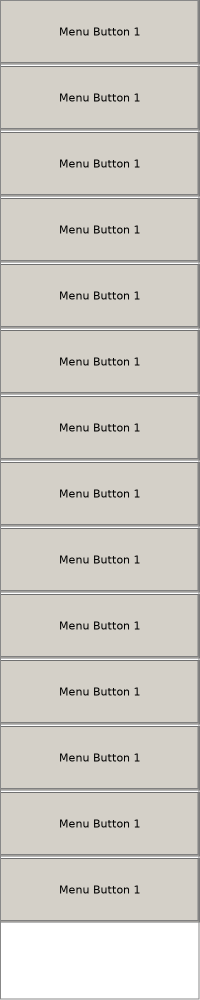
VISUALIZATION PopupMenu1  // 200x1000
    Button (0,0 200x64), "Menu Button 1"
    Button (0,66 200x64), "Menu Button 1"
    Button (0,132 200x64), "Menu Button 1"
    Button (0,198 200x64), "Menu Button 1"
    Button (0,264 200x64), "Menu Button 1"
    Button (0,330 200x64), "Menu Button 1"
    Button (0,396 200x64), "Menu Button 1"
    Button (0,462 200x64), "Menu Button 1"
    Button (0,528 200x64), "Menu Button 1"
    Button (0,594 200x64), "Menu Button 1"
    Button (0,660 200x64), "Menu Button 1"
    Button (0,726 200x64), "Menu Button 1"
    Button (0,792 200x64), "Menu Button 1"
    Button (0,858 200x64), "Menu Button 1"
END_VISUALIZATION

(* stored: Version 1.1.0.1, ProductVersion 3.1.4024.11
   Visu PopupMenu1: Id {583ba4a9-9f28-0dc2-1a95-a2c16aeb563e} *)
